TYPE COLLECTION_INDEX : DINT(0..2147483647 - 1); END_TYPE

(* stored: Version 1.1.0.1
   DUT COLLECTION_INDEX: Id {cb31a08b-1d48-441f-ae8b-ce1d5fc80f31} *)
